// TIA Portal V20 export
DATA_BLOCK "DB_WarmUP"   // DB530
// stored: AutoNumber false, InstanceOfName FB_WarmUP, InstanceOfType FB
"FB_WarmUP"
   // VAR
   //    sWarmUpTimer : Time;
   //    sLimitedWarmupTime : Bool;
   //    sUnlimitedWarmupTime : Bool;
   //    sActualWarmupTime : Time;
   //    sRemainingWarmupMinutes : Int;
   //    sDeltaTimeWarmup : Time;
   //    sLimitedWarmUP : TON_TIME;
   //    sStartWarmup { S7_SetPoint := 'True'} : Bool;
   //    sUnlimitedWarmUP : TON_TIME;
   //    sUnlimitedWarmUPCounter { S7_SetPoint := 'True'} : "FB_TimeCounter";
   // END_VAR
BEGIN
END_DATA_BLOCK
